VAR_GLOBAL
	currentOrderData	:	OrderData;
	nextJobReady	:	BOOL;
	reOrderDone	:	R_TRIG;
	reNewOrderSend	:	R_TRIG;
	reShiftSerialNumber	:	R_TRIG;
END_VAR

(* stored: Version 1.1.0.1
   GVL OrderManagement: Id {3d1cffef-548e-4995-89bf-e9fb4ff0ce2e} *)
